FUNCTION_BLOCK TTestEventHandler IMPLEMENTS ITestEventHandler
VAR
    _EventWasRaised : BOOL;
    _EventData : UDINT;
END_VAR

PROPERTY EventWasRaised : BOOL
GET
EventWasRaised := _EventWasRaised;
END_GET
END_PROPERTY

METHOD OnCustomEvent
VAR_INPUT
    EventData : UDINT;
END_VAR
_EventData := EventData;
_EventWasRaised := TRUE;
END_METHOD

END_FUNCTION_BLOCK

(* stored: Version 1.1.0.1, ProductVersion 3.1.4024.3
   POU TTestEventHandler: Id {6a7e5cff-3f08-4226-848e-9c6f81658547}, SpecialFunc None
   Property EventWasRaised: Id {7a1929c0-2d78-4ce8-a7ba-9401c0f26865}
   Get Get: Id {a1df0a15-f7f1-4fd4-893f-6b128e9e5c1b}
   Method OnCustomEvent: Id {d6e5babe-d6eb-4995-8c07-2c5fc8c98c96} *)
